PROGRAM Motors_Speed_IO
VAR_OUTPUT
	//Values to send to the motors
	fToSend1 : REAL;
	fToSend2 : REAL;
	fToSend3 : REAL;
	fToSend4 : REAL;
	
	//Booleans confirming that something has been sent...
	bSend1Ready : BOOL := FALSE;
	bSend2Ready : BOOL := FALSE;
	bSend3Ready : BOOL := FALSE;
	bSend4Ready : BOOL := FALSE;
END_VAR

VAR
	R_TRIG_0: R_TRIG;
	R_TRIG_1: R_TRIG;
	R_TRIG_2: R_TRIG;
	R_TRIG_3: R_TRIG;
END_VAR
VAR // added by the converter: edge detectors and wires of the graphical bodies
    _w1, _w2, _w3, _w4 : BOOL;
END_VAR

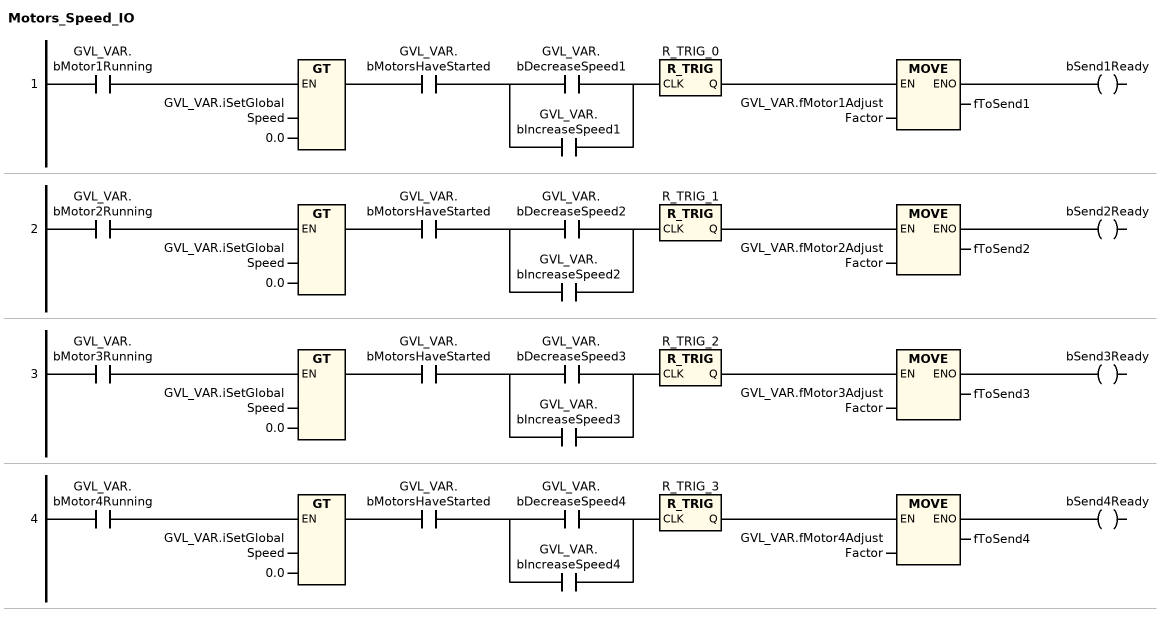
// NETWORK 1
R_TRIG_0(CLK := (GVL_VAR.bMotor1Running AND GVL_VAR.iSetGlobalSpeed > 0.0) AND GVL_VAR.bMotorsHaveStarted AND (GVL_VAR.bDecreaseSpeed1 OR GVL_VAR.bIncreaseSpeed1)); // R_TRIG
_w1 := R_TRIG_0.Q;
IF _w1 THEN fToSend1 := GVL_VAR.fMotor1AdjustFactor; END_IF
bSend1Ready := _w1;

// NETWORK 2
R_TRIG_1(CLK := (GVL_VAR.bMotor2Running AND GVL_VAR.iSetGlobalSpeed > 0.0) AND GVL_VAR.bMotorsHaveStarted AND (GVL_VAR.bDecreaseSpeed2 OR GVL_VAR.bIncreaseSpeed2)); // R_TRIG
_w2 := R_TRIG_1.Q;
IF _w2 THEN fToSend2 := GVL_VAR.fMotor2AdjustFactor; END_IF
bSend2Ready := _w2;

// NETWORK 3
R_TRIG_2(CLK := (GVL_VAR.bMotor3Running AND GVL_VAR.iSetGlobalSpeed > 0.0) AND GVL_VAR.bMotorsHaveStarted AND (GVL_VAR.bDecreaseSpeed3 OR GVL_VAR.bIncreaseSpeed3)); // R_TRIG
_w3 := R_TRIG_2.Q;
IF _w3 THEN fToSend3 := GVL_VAR.fMotor3AdjustFactor; END_IF
bSend3Ready := _w3;

// NETWORK 4
R_TRIG_3(CLK := (GVL_VAR.bMotor4Running AND GVL_VAR.iSetGlobalSpeed > 0.0) AND GVL_VAR.bMotorsHaveStarted AND (GVL_VAR.bDecreaseSpeed4 OR GVL_VAR.bIncreaseSpeed4)); // R_TRIG
_w4 := R_TRIG_3.Q;
IF _w4 THEN fToSend4 := GVL_VAR.fMotor4AdjustFactor; END_IF
bSend4Ready := _w4;

END_PROGRAM

(* stored: Version 1.1.0.1, ProductVersion 3.1.4024.12
   POU Motors_Speed_IO: Id {85a3b94c-1f5b-40a9-a31d-dded3793d71b}, SpecialFunc None *)
